TEXTLIST TL_Mparams_LREAL
  1 = 'AbsoluteHigh'
  2 = 'AbsoluteLow'
  3 = 'ExtruderComp'
  4 = 'KpCool'
  5 = 'KpHeat'
  6 = 'TdCool'
  7 = 'TdHeat'
  8 = 'TnCool'
  9 = 'TnHeat'
  10 = 'TvCool'
  11 = 'TvHeat'
  12 = 'Overshoot'
  13 = 'Tracking_Rate'
  14 = 'Tracking_Td'
  15 = 'Ramping_Rate'
  16 = 'Ramping_RateC'
  17 = 'Ramping_Tolerance'
  18 = 'dTmax'
  19 = 'SensorOffset'
  20 = 'SettlingTime'
  21 = 'SupplyLoad_Cooler'
  22 = 'SupplyLoad_Heater'
  23 = 'SupplyLoad_Tolerance'
  24 = 'TuneEnd'
  25 = 'TuneKp'
  26 = 'TuneTd'
  27 = 'TuneTn'
  28 = 'TuneTv'
  29 = 'TuneTrackingTd'
  30 = 'TuneY'
  31 = 'L_LoadIdle'
  32 = 'Weighting_C'
  33 = 'ErrorHeatingFactor'
  34 = 'fPwmStdMaxOnTime'
  35 = '*** not Used ***'
  36 = 'fPwmMinOnTime'
  37 = 'fc_OnTime'
  38 = 'fc_OffTime'
  39 = 'ActTempGain'
  40 = 'ActTempOffset'
  41 = 'SaveDelay'
   = ''
END_TEXTLIST

(* stored: Version 1.1.0.1, ProductVersion 3.1.4020.12
   TextList TL_Mparams_LREAL: Id {113a79a4-34f1-45a8-8172-4a3b875c83b4} *)
